// Mitsubishi GX Works2 project: PROGRAMA CLP   PLC: FX3U/FX3UC
// Configuração Modbus RTU

PROGRAM MAIN
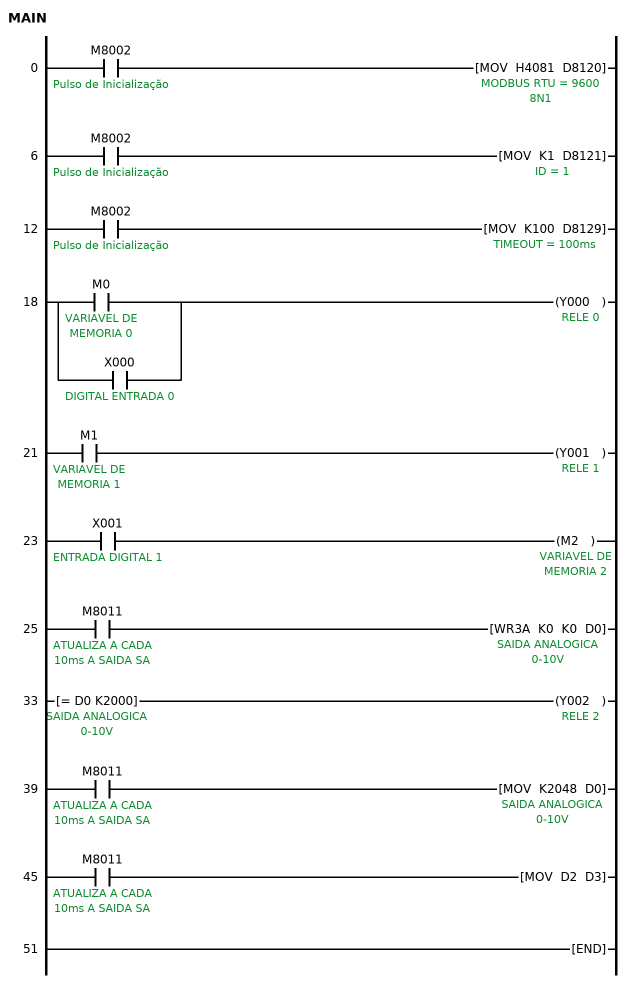
0     LD      M8002  ; Pulso de Inicialização
      MOV     H4081 D8120  ; MODBUS RTU = 9600 8N1
6     LD      M8002  ; Pulso de Inicialização
      MOV     K1 D8121  ; ID = 1
12    LD      M8002  ; Pulso de Inicialização
      MOV     K100 D8129  ; TIMEOUT = 100ms
18    LD      M0  ; VARIAVEL DE MEMORIA 0
      OR      X000  ; DIGITAL ENTRADA 0
      OUT     Y000  ; RELE 0
21    LD      M1  ; VARIAVEL DE MEMORIA 1
      OUT     Y001  ; RELE 1
23    LD      X001  ; ENTRADA DIGITAL 1
      OUT     M2  ; VARIAVEL DE MEMORIA 2
25    LD      M8011  ; ATUALIZA A CADA 10ms A SAIDA SA
      WR3A    K0 K0 D0  ; SAIDA ANALOGICA 0-10V
33    LD=     D0 K2000  ; SAIDA ANALOGICA 0-10V
      OUT     Y002  ; RELE 2
39    LD      M8011  ; ATUALIZA A CADA 10ms A SAIDA SA
      MOV     K2048 D0
45    LD      M8011  ; ATUALIZA A CADA 10ms A SAIDA SA
      MOV     D2 D3
51    END
END_PROGRAM
